TYPE Out_16_To_PLC :
STRUCT
	Out AT %I*:ARRAY [1..16] OF BOOL;
END_STRUCT
END_TYPE

(* stored: Version 1.1.0.1, ProductVersion 3.1.4024.14
   DUT Out_16_To_PLC: Id {08bcfaac-d822-4a69-84a1-655efc106331} *)
